{attribute 'qualified_only'}
{attribute 'strict'}
TYPE E_DbLogState :
(
    idle := 0,
    init,
    writing,
    error
);
END_TYPE

(* stored: Version 1.1.0.1, ProductVersion 3.1.4024.9
   DUT E_DbLogState: Id {e7a4300f-5312-4ae7-a2ad-554daf4e1440} *)
